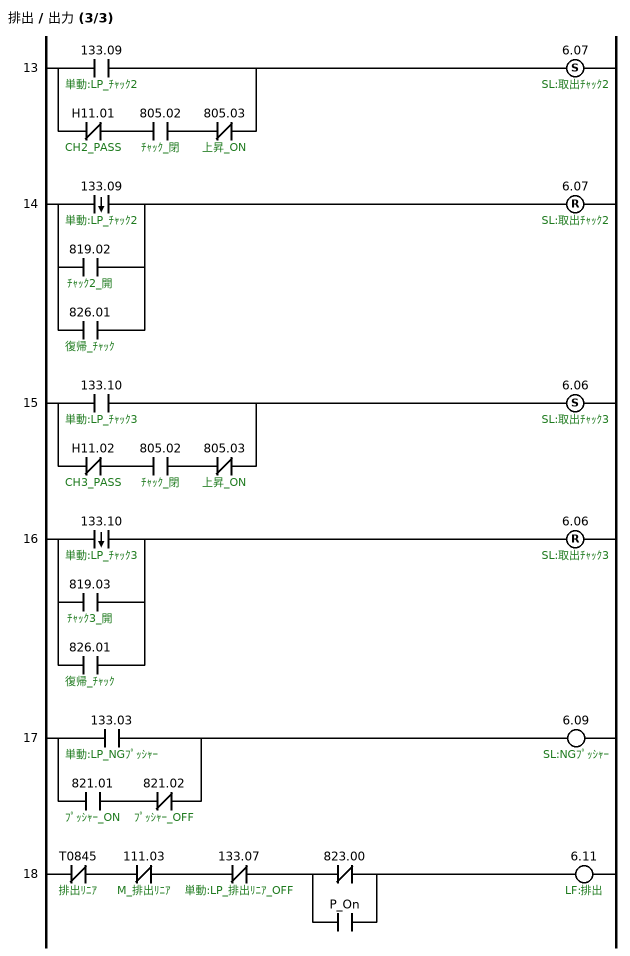
; [picture p192: 排出 / 出力, rungs 13-18]
; rung 13
LD 133.09  ; 単動:LP_ﾁｬｯｸ2
LDNOT H11.01  ; CH2_PASS
AND 805.02  ; ﾁｬｯｸ_閉
ANDNOT 805.03  ; 上昇_ON
ORLD
SET 6.07  ; SL:取出ﾁｬｯｸ2
; rung 14
%LD 133.09  ; 単動:LP_ﾁｬｯｸ2
OR 819.02  ; ﾁｬｯｸ2_開
OR 826.01  ; 復帰_ﾁｬｯｸ
RSET 6.07  ; SL:取出ﾁｬｯｸ2
; rung 15
LD 133.10  ; 単動:LP_ﾁｬｯｸ3
LDNOT H11.02  ; CH3_PASS
AND 805.02  ; ﾁｬｯｸ_閉
ANDNOT 805.03  ; 上昇_ON
ORLD
SET 6.06  ; SL:取出ﾁｬｯｸ3
; rung 16
%LD 133.10  ; 単動:LP_ﾁｬｯｸ3
OR 819.03  ; ﾁｬｯｸ3_開
OR 826.01  ; 復帰_ﾁｬｯｸ
RSET 6.06  ; SL:取出ﾁｬｯｸ3
; rung 17
LD 133.03  ; 単動:LP_NGﾌﾟｯｼｬｰ
LD 821.01  ; ﾌﾟｯｼｬｰ_ON
ANDNOT 821.02  ; ﾌﾟｯｼｬｰ_OFF
ORLD
OUT 6.09  ; SL:NGﾌﾟｯｼｬｰ
; rung 18
LDNOT T0845  ; 排出ﾘﾆｱ
ANDNOT 111.03  ; M_排出ﾘﾆｱ
ANDNOT 133.07  ; 単動:LP_排出ﾘﾆｱ_OFF
LDNOT 823.00
OR P_On
ANDLD
OUT 6.11  ; LF:排出

### Section ｴﾗｰ

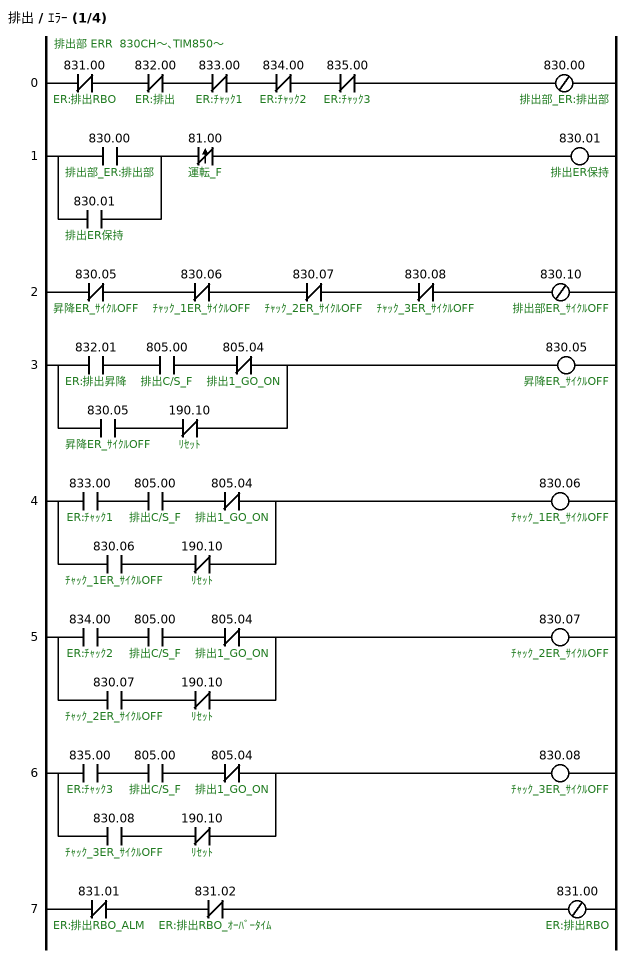
; rung 0: 排出部 ERR  830CH～､TIM850～
LDNOT 831.00  ; ER:排出RBO
ANDNOT 832.00  ; ER:排出
ANDNOT 833.00  ; ER:ﾁｬｯｸ1
ANDNOT 834.00  ; ER:ﾁｬｯｸ2
ANDNOT 835.00  ; ER:ﾁｬｯｸ3
OUTNOT 830.00  ; 排出部_ER:排出部
; rung 1
LD 830.00  ; 排出部_ER:排出部
OR 830.01  ; 排出ER保持
@ANDNOT 81.00  ; 運転_F
OUT 830.01  ; 排出ER保持
; rung 2
LDNOT 830.05  ; 昇降ER_ｻｲｸﾙOFF
ANDNOT 830.06  ; ﾁｬｯｸ_1ER_ｻｲｸﾙOFF
ANDNOT 830.07  ; ﾁｬｯｸ_2ER_ｻｲｸﾙOFF
ANDNOT 830.08  ; ﾁｬｯｸ_3ER_ｻｲｸﾙOFF
OUTNOT 830.10  ; 排出部ER_ｻｲｸﾙOFF
; rung 3
LD 832.01  ; ER:排出昇降
AND 805.00  ; 排出C/S_F
ANDNOT 805.04  ; 排出1_GO_ON
LD 830.05  ; 昇降ER_ｻｲｸﾙOFF
ANDNOT 190.10  ; ﾘｾｯﾄ
ORLD
OUT 830.05  ; 昇降ER_ｻｲｸﾙOFF
; rung 4
LD 833.00  ; ER:ﾁｬｯｸ1
AND 805.00  ; 排出C/S_F
ANDNOT 805.04  ; 排出1_GO_ON
LD 830.06  ; ﾁｬｯｸ_1ER_ｻｲｸﾙOFF
ANDNOT 190.10  ; ﾘｾｯﾄ
ORLD
OUT 830.06  ; ﾁｬｯｸ_1ER_ｻｲｸﾙOFF
; rung 5
LD 834.00  ; ER:ﾁｬｯｸ2
AND 805.00  ; 排出C/S_F
ANDNOT 805.04  ; 排出1_GO_ON
LD 830.07  ; ﾁｬｯｸ_2ER_ｻｲｸﾙOFF
ANDNOT 190.10  ; ﾘｾｯﾄ
ORLD
OUT 830.07  ; ﾁｬｯｸ_2ER_ｻｲｸﾙOFF
; rung 6
LD 835.00  ; ER:ﾁｬｯｸ3
AND 805.00  ; 排出C/S_F
ANDNOT 805.04  ; 排出1_GO_ON
LD 830.08  ; ﾁｬｯｸ_3ER_ｻｲｸﾙOFF
ANDNOT 190.10  ; ﾘｾｯﾄ
ORLD
OUT 830.08  ; ﾁｬｯｸ_3ER_ｻｲｸﾙOFF
; rung 7
LDNOT 831.01  ; ER:排出RBO_ALM
ANDNOT 831.02  ; ER:排出RBO_ｵｰﾊﾞｰﾀｲﾑ
OUTNOT 831.00  ; ER:排出RBO

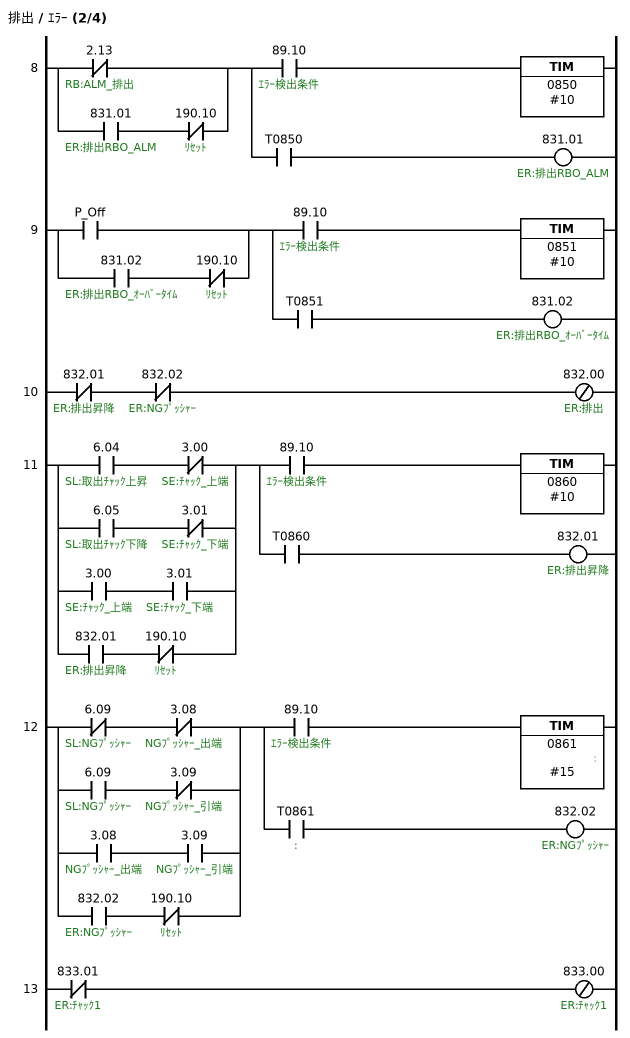
; rung 8
LDNOT 2.13  ; RB:ALM_排出
LD 831.01  ; ER:排出RBO_ALM
ANDNOT 190.10  ; ﾘｾｯﾄ
ORLD
OUT TR0
AND 89.10  ; ｴﾗｰ検出条件
TIM 0850 #10
LD TR0
AND T0850
OUT 831.01  ; ER:排出RBO_ALM
; rung 9
LD P_Off
LD 831.02  ; ER:排出RBO_ｵｰﾊﾞｰﾀｲﾑ
ANDNOT 190.10  ; ﾘｾｯﾄ
ORLD
OUT TR0
AND 89.10  ; ｴﾗｰ検出条件
TIM 0851 #10
LD TR0
AND T0851
OUT 831.02  ; ER:排出RBO_ｵｰﾊﾞｰﾀｲﾑ
; rung 10
LDNOT 832.01  ; ER:排出昇降
ANDNOT 832.02  ; ER:NGﾌﾟｯｼｬｰ
OUTNOT 832.00  ; ER:排出
; rung 11
LD 6.04  ; SL:取出ﾁｬｯｸ上昇
ANDNOT 3.00  ; SE:ﾁｬｯｸ_上端
LD 6.05  ; SL:取出ﾁｬｯｸ下降
ANDNOT 3.01  ; SE:ﾁｬｯｸ_下端
ORLD
LD 3.00  ; SE:ﾁｬｯｸ_上端
AND 3.01  ; SE:ﾁｬｯｸ_下端
ORLD
LD 832.01  ; ER:排出昇降
ANDNOT 190.10  ; ﾘｾｯﾄ
ORLD
OUT TR0
AND 89.10  ; ｴﾗｰ検出条件
TIM 0860 #10
LD TR0
AND T0860
OUT 832.01  ; ER:排出昇降
; rung 12
LDNOT 6.09  ; SL:NGﾌﾟｯｼｬｰ
ANDNOT 3.08  ; NGﾌﾟｯｼｬｰ_出端
LD 6.09  ; SL:NGﾌﾟｯｼｬｰ
ANDNOT 3.09  ; NGﾌﾟｯｼｬｰ_引端
ORLD
LD 3.08  ; NGﾌﾟｯｼｬｰ_出端
AND 3.09  ; NGﾌﾟｯｼｬｰ_引端
ORLD
LD 832.02  ; ER:NGﾌﾟｯｼｬｰ
ANDNOT 190.10  ; ﾘｾｯﾄ
ORLD
OUT TR0
AND 89.10  ; ｴﾗｰ検出条件
TIM 0861 #15  ; :
LD TR0
AND T0861  ; :
OUT 832.02  ; ER:NGﾌﾟｯｼｬｰ
; rung 13
LDNOT 833.01  ; ER:ﾁｬｯｸ1
OUTNOT 833.00  ; ER:ﾁｬｯｸ1

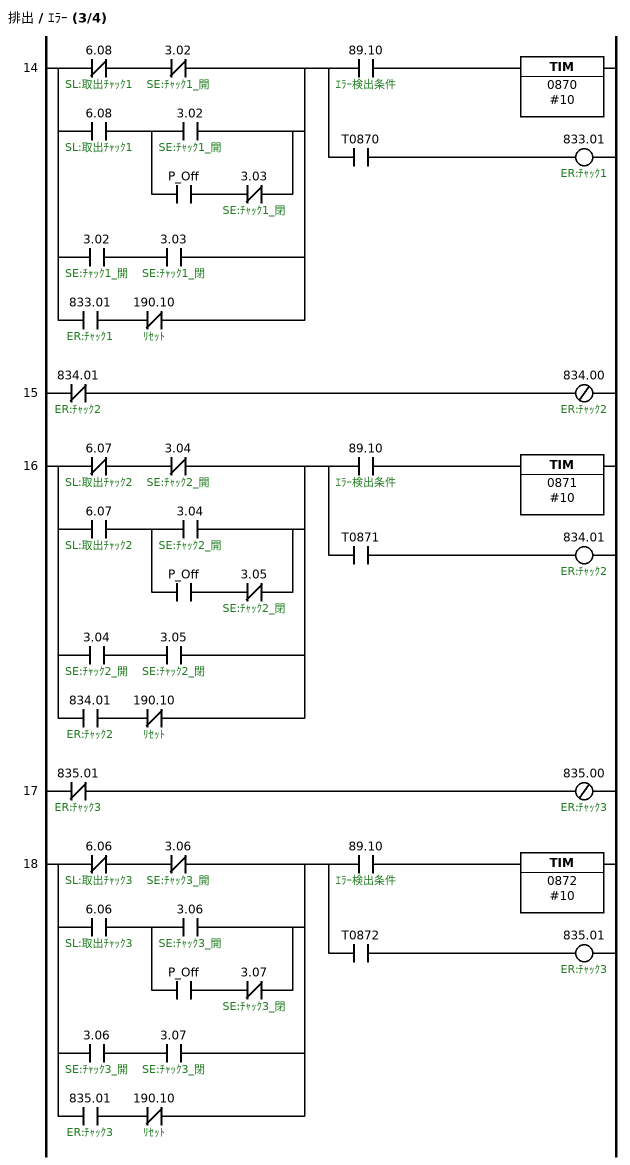
; rung 14
LDNOT 6.08  ; SL:取出ﾁｬｯｸ1
ANDNOT 3.02  ; SE:ﾁｬｯｸ1_開
LD 6.08  ; SL:取出ﾁｬｯｸ1
LD 3.02  ; SE:ﾁｬｯｸ1_開
LD P_Off
ANDNOT 3.03  ; SE:ﾁｬｯｸ1_閉
ORLD
ANDLD
ORLD
LD 3.02  ; SE:ﾁｬｯｸ1_開
AND 3.03  ; SE:ﾁｬｯｸ1_閉
ORLD
LD 833.01  ; ER:ﾁｬｯｸ1
ANDNOT 190.10  ; ﾘｾｯﾄ
ORLD
OUT TR0
AND 89.10  ; ｴﾗｰ検出条件
TIM 0870 #10
LD TR0
AND T0870
OUT 833.01  ; ER:ﾁｬｯｸ1
; rung 15
LDNOT 834.01  ; ER:ﾁｬｯｸ2
OUTNOT 834.00  ; ER:ﾁｬｯｸ2
; rung 16
LDNOT 6.07  ; SL:取出ﾁｬｯｸ2
ANDNOT 3.04  ; SE:ﾁｬｯｸ2_開
LD 6.07  ; SL:取出ﾁｬｯｸ2
LD 3.04  ; SE:ﾁｬｯｸ2_開
LD P_Off
ANDNOT 3.05  ; SE:ﾁｬｯｸ2_閉
ORLD
ANDLD
ORLD
LD 3.04  ; SE:ﾁｬｯｸ2_開
AND 3.05  ; SE:ﾁｬｯｸ2_閉
ORLD
LD 834.01  ; ER:ﾁｬｯｸ2
ANDNOT 190.10  ; ﾘｾｯﾄ
ORLD
OUT TR0
AND 89.10  ; ｴﾗｰ検出条件
TIM 0871 #10
LD TR0
AND T0871
OUT 834.01  ; ER:ﾁｬｯｸ2
; rung 17
LDNOT 835.01  ; ER:ﾁｬｯｸ3
OUTNOT 835.00  ; ER:ﾁｬｯｸ3
; rung 18
LDNOT 6.06  ; SL:取出ﾁｬｯｸ3
ANDNOT 3.06  ; SE:ﾁｬｯｸ3_開
LD 6.06  ; SL:取出ﾁｬｯｸ3
LD 3.06  ; SE:ﾁｬｯｸ3_開
LD P_Off
ANDNOT 3.07  ; SE:ﾁｬｯｸ3_閉
ORLD
ANDLD
ORLD
LD 3.06  ; SE:ﾁｬｯｸ3_開
AND 3.07  ; SE:ﾁｬｯｸ3_閉
ORLD
LD 835.01  ; ER:ﾁｬｯｸ3
ANDNOT 190.10  ; ﾘｾｯﾄ
ORLD
OUT TR0
AND 89.10  ; ｴﾗｰ検出条件
TIM 0872 #10
LD TR0
AND T0872
OUT 835.01  ; ER:ﾁｬｯｸ3

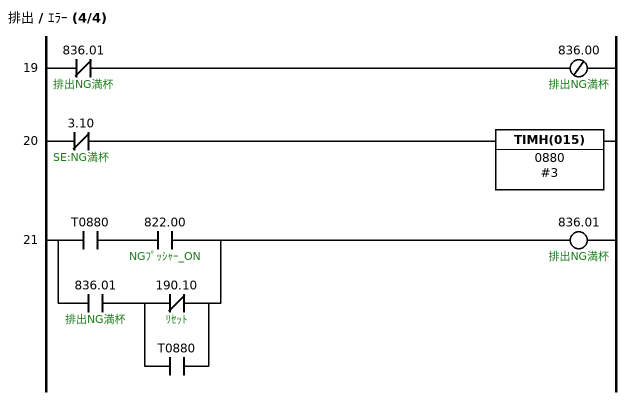
; rung 19
LDNOT 836.01  ; 排出NG満杯
OUTNOT 836.00  ; 排出NG満杯
; rung 20
LDNOT 3.10  ; SE:NG満杯
TIMH(015) 0880 #3
; rung 21
LD T0880
AND 822.00  ; NGﾌﾟｯｼｬｰ_ON
LD 836.01  ; 排出NG満杯
LDNOT 190.10  ; ﾘｾｯﾄ
OR T0880
ANDLD
ORLD
OUT 836.01  ; 排出NG満杯

### Section END
; rung 0
END(001)

## Program ﾃﾞｰﾀ収集 (cyclic task 8)

### Section 通信ST

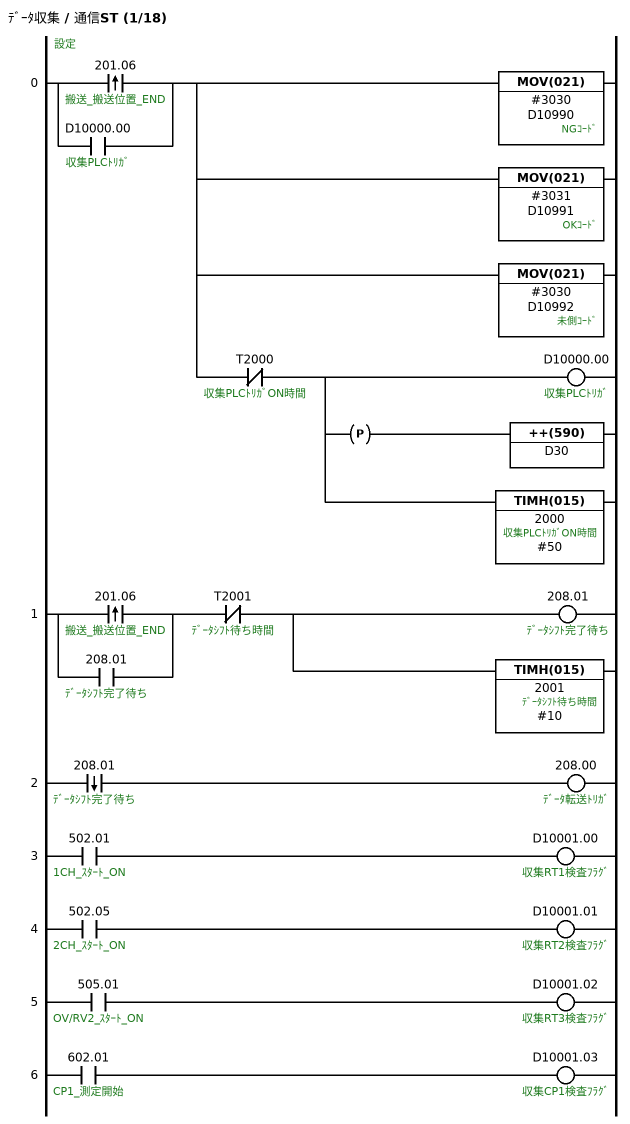
; rung 0: 設定
@LD 201.06  ; 搬送_搬送位置_END
OR D10000.00  ; 収集PLCﾄﾘｶﾞ
MOV(021) #3030 D10990  ; NGｺｰﾄﾞ
MOV(021) #3031 D10991  ; OKｺｰﾄﾞ
MOV(021) #3030 D10992  ; 未側ｺｰﾄﾞ
ANDNOT T2000  ; 収集PLCﾄﾘｶﾞON時間
OUT TR0
OUT D10000.00  ; 収集PLCﾄﾘｶﾞ
UP(521)
++(590) D30
LD TR0
TIMH(015) 2000 #50  ; 収集PLCﾄﾘｶﾞON時間
; rung 1
@LD 201.06  ; 搬送_搬送位置_END
OR 208.01  ; ﾃﾞｰﾀｼﾌﾄ完了待ち
ANDNOT T2001  ; ﾃﾞｰﾀｼﾌﾄ待ち時間
OUT 208.01  ; ﾃﾞｰﾀｼﾌﾄ完了待ち
TIMH(015) 2001 #10  ; ﾃﾞｰﾀｼﾌﾄ待ち時間
; rung 2
%LD 208.01  ; ﾃﾞｰﾀｼﾌﾄ完了待ち
OUT 208.00  ; ﾃﾞｰﾀ転送ﾄﾘｶﾞ
; rung 3
LD 502.01  ; 1CH_ｽﾀｰﾄ_ON
OUT D10001.00  ; 収集RT1検査ﾌﾗｸﾞ
; rung 4
LD 502.05  ; 2CH_ｽﾀｰﾄ_ON
OUT D10001.01  ; 収集RT2検査ﾌﾗｸﾞ
; rung 5
LD 505.01  ; OV/RV2_ｽﾀｰﾄ_ON
OUT D10001.02  ; 収集RT3検査ﾌﾗｸﾞ
; rung 6
LD 602.01  ; CP1_測定開始
OUT D10001.03  ; 収集CP1検査ﾌﾗｸﾞ

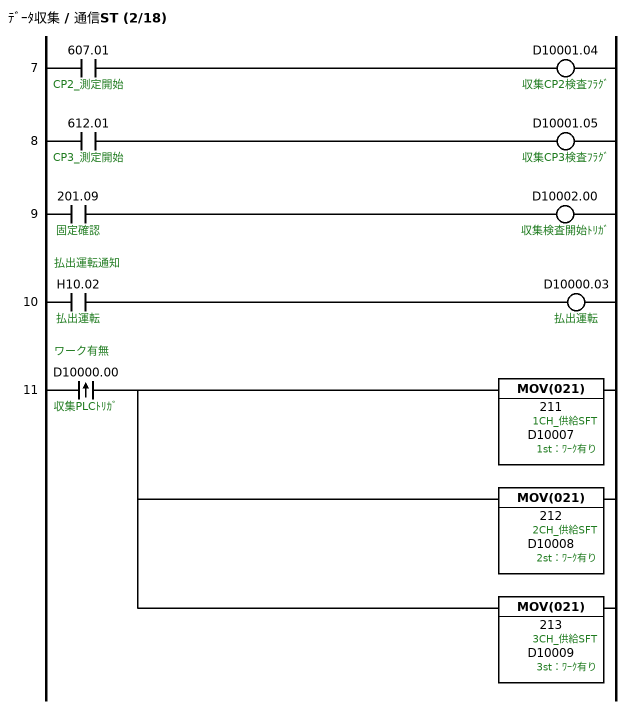
; rung 7
LD 607.01  ; CP2_測定開始
OUT D10001.04  ; 収集CP2検査ﾌﾗｸﾞ
; rung 8
LD 612.01  ; CP3_測定開始
OUT D10001.05  ; 収集CP3検査ﾌﾗｸﾞ
; rung 9
LD 201.09  ; 固定確認
OUT D10002.00  ; 収集検査開始ﾄﾘｶﾞ
; rung 10: 払出運転通知
LD H10.02  ; 払出運転
OUT D10000.03  ; 払出運転
; rung 11: ワーク有無
@LD D10000.00  ; 収集PLCﾄﾘｶﾞ
MOV(021) 211 D10007  ; 1CH_供給SFT, 1st：ﾜｰｸ有り
MOV(021) 212 D10008  ; 2CH_供給SFT, 2st：ﾜｰｸ有り
MOV(021) 213 D10009  ; 3CH_供給SFT, 3st：ﾜｰｸ有り

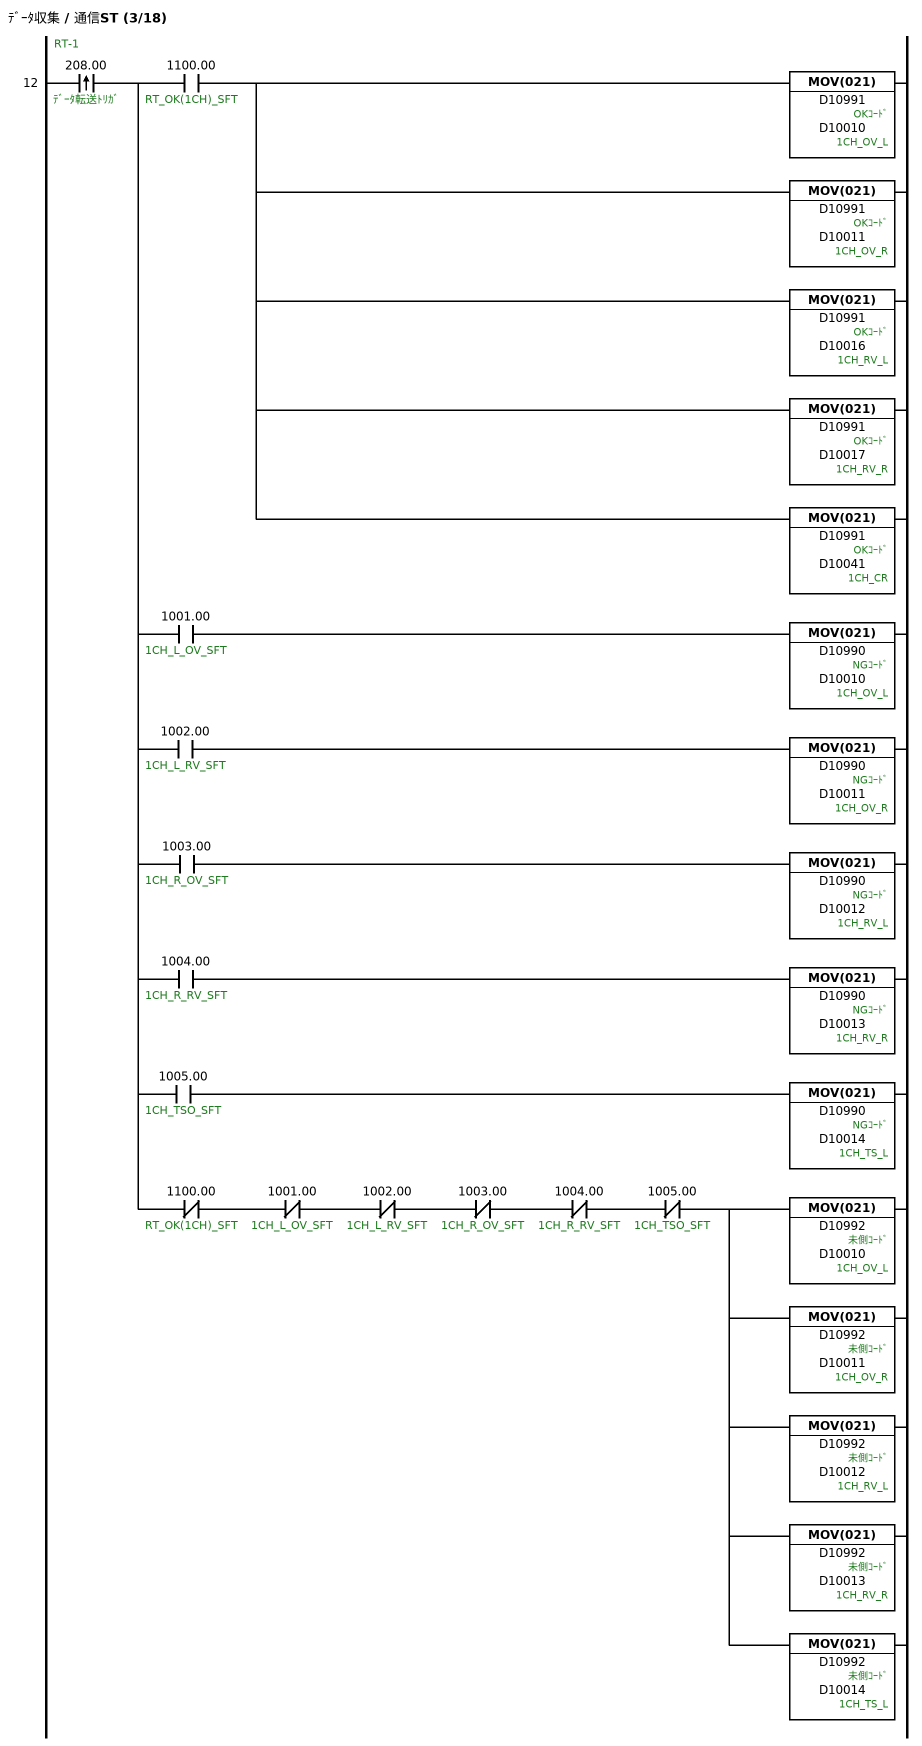
; rung 12: RT-1
@LD 208.00  ; ﾃﾞｰﾀ転送ﾄﾘｶﾞ
OUT TR0
AND 1100.00  ; RT_OK(1CH)_SFT
MOV(021) D10991 D10010  ; OKｺｰﾄﾞ, 1CH_OV_L
MOV(021) D10991 D10011  ; OKｺｰﾄﾞ, 1CH_OV_R
MOV(021) D10991 D10016  ; OKｺｰﾄﾞ, 1CH_RV_L
MOV(021) D10991 D10017  ; OKｺｰﾄﾞ, 1CH_RV_R
MOV(021) D10991 D10041  ; OKｺｰﾄﾞ, 1CH_CR
LD TR0
AND 1001.00  ; 1CH_L_OV_SFT
MOV(021) D10990 D10010  ; NGｺｰﾄﾞ, 1CH_OV_L
LD TR0
AND 1002.00  ; 1CH_L_RV_SFT
MOV(021) D10990 D10011  ; NGｺｰﾄﾞ, 1CH_OV_R
LD TR0
AND 1003.00  ; 1CH_R_OV_SFT
MOV(021) D10990 D10012  ; NGｺｰﾄﾞ, 1CH_RV_L
LD TR0
AND 1004.00  ; 1CH_R_RV_SFT
MOV(021) D10990 D10013  ; NGｺｰﾄﾞ, 1CH_RV_R
LD TR0
AND 1005.00  ; 1CH_TSO_SFT
MOV(021) D10990 D10014  ; NGｺｰﾄﾞ, 1CH_TS_L
LD TR0
ANDNOT 1100.00  ; RT_OK(1CH)_SFT
ANDNOT 1001.00  ; 1CH_L_OV_SFT
ANDNOT 1002.00  ; 1CH_L_RV_SFT
ANDNOT 1003.00  ; 1CH_R_OV_SFT
ANDNOT 1004.00  ; 1CH_R_RV_SFT
ANDNOT 1005.00  ; 1CH_TSO_SFT
MOV(021) D10992 D10010  ; 未側ｺｰﾄﾞ, 1CH_OV_L
MOV(021) D10992 D10011  ; 未側ｺｰﾄﾞ, 1CH_OV_R
MOV(021) D10992 D10012  ; 未側ｺｰﾄﾞ, 1CH_RV_L
MOV(021) D10992 D10013  ; 未側ｺｰﾄﾞ, 1CH_RV_R
MOV(021) D10992 D10014  ; 未側ｺｰﾄﾞ, 1CH_TS_L

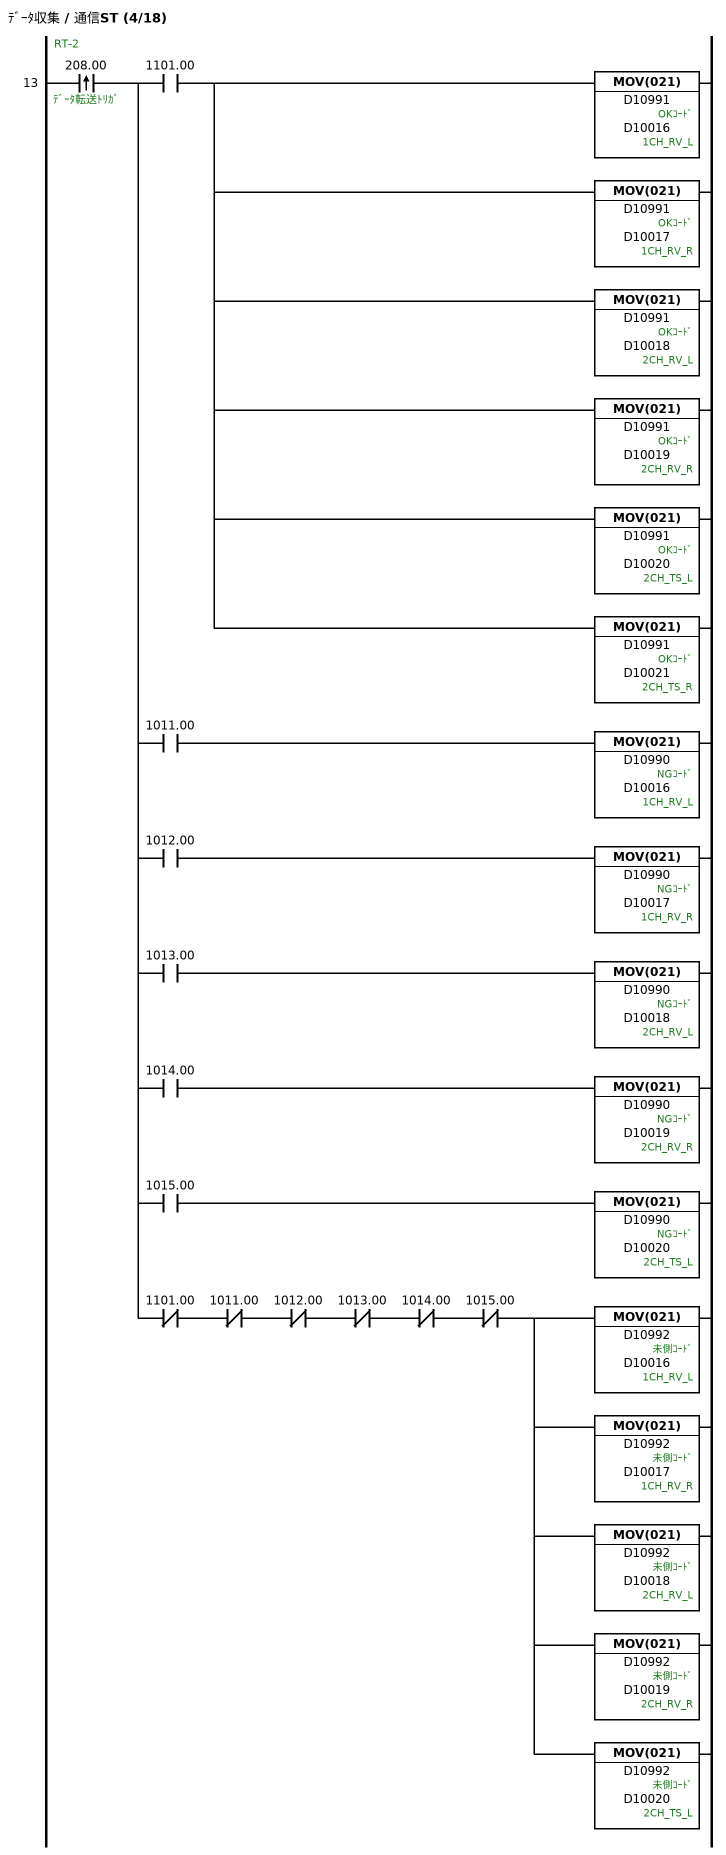
; rung 13: RT-2
@LD 208.00  ; ﾃﾞｰﾀ転送ﾄﾘｶﾞ
OUT TR0
AND 1101.00
MOV(021) D10991 D10016  ; OKｺｰﾄﾞ, 1CH_RV_L
MOV(021) D10991 D10017  ; OKｺｰﾄﾞ, 1CH_RV_R
MOV(021) D10991 D10018  ; OKｺｰﾄﾞ, 2CH_RV_L
MOV(021) D10991 D10019  ; OKｺｰﾄﾞ, 2CH_RV_R
MOV(021) D10991 D10020  ; OKｺｰﾄﾞ, 2CH_TS_L
MOV(021) D10991 D10021  ; OKｺｰﾄﾞ, 2CH_TS_R
LD TR0
AND 1011.00
MOV(021) D10990 D10016  ; NGｺｰﾄﾞ, 1CH_RV_L
LD TR0
AND 1012.00
MOV(021) D10990 D10017  ; NGｺｰﾄﾞ, 1CH_RV_R
LD TR0
AND 1013.00
MOV(021) D10990 D10018  ; NGｺｰﾄﾞ, 2CH_RV_L
LD TR0
AND 1014.00
MOV(021) D10990 D10019  ; NGｺｰﾄﾞ, 2CH_RV_R
LD TR0
AND 1015.00
MOV(021) D10990 D10020  ; NGｺｰﾄﾞ, 2CH_TS_L
LD TR0
ANDNOT 1101.00
ANDNOT 1011.00
ANDNOT 1012.00
ANDNOT 1013.00
ANDNOT 1014.00
ANDNOT 1015.00
MOV(021) D10992 D10016  ; 未側ｺｰﾄﾞ, 1CH_RV_L
MOV(021) D10992 D10017  ; 未側ｺｰﾄﾞ, 1CH_RV_R
MOV(021) D10992 D10018  ; 未側ｺｰﾄﾞ, 2CH_RV_L
MOV(021) D10992 D10019  ; 未側ｺｰﾄﾞ, 2CH_RV_R
MOV(021) D10992 D10020  ; 未側ｺｰﾄﾞ, 2CH_TS_L

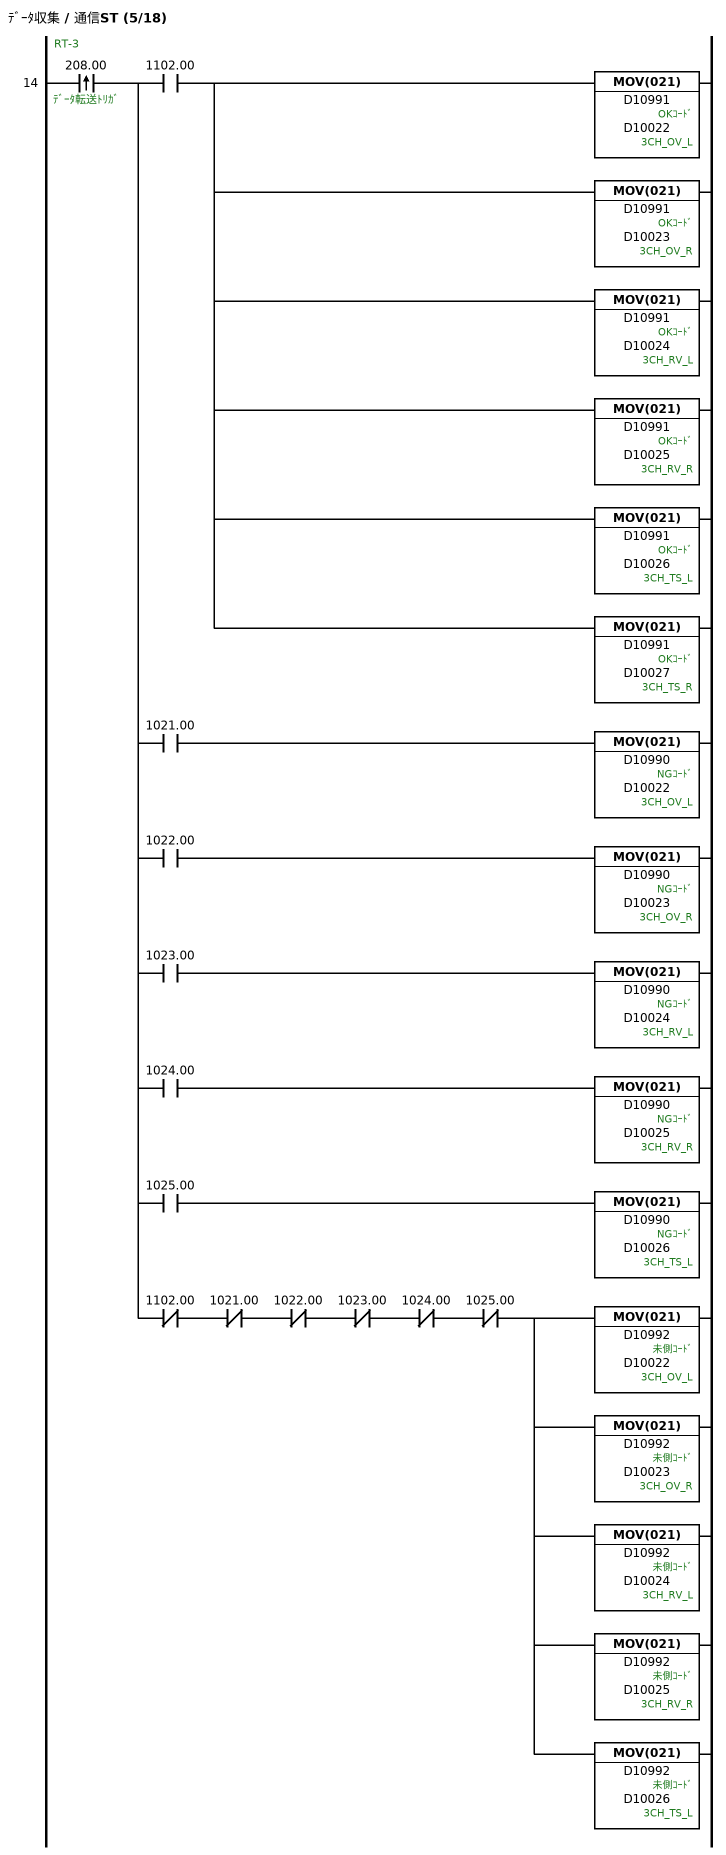
; rung 14: RT-3
@LD 208.00  ; ﾃﾞｰﾀ転送ﾄﾘｶﾞ
OUT TR0
AND 1102.00
MOV(021) D10991 D10022  ; OKｺｰﾄﾞ, 3CH_OV_L
MOV(021) D10991 D10023  ; OKｺｰﾄﾞ, 3CH_OV_R
MOV(021) D10991 D10024  ; OKｺｰﾄﾞ, 3CH_RV_L
MOV(021) D10991 D10025  ; OKｺｰﾄﾞ, 3CH_RV_R
MOV(021) D10991 D10026  ; OKｺｰﾄﾞ, 3CH_TS_L
MOV(021) D10991 D10027  ; OKｺｰﾄﾞ, 3CH_TS_R
LD TR0
AND 1021.00
MOV(021) D10990 D10022  ; NGｺｰﾄﾞ, 3CH_OV_L
LD TR0
AND 1022.00
MOV(021) D10990 D10023  ; NGｺｰﾄﾞ, 3CH_OV_R
LD TR0
AND 1023.00
MOV(021) D10990 D10024  ; NGｺｰﾄﾞ, 3CH_RV_L
LD TR0
AND 1024.00
MOV(021) D10990 D10025  ; NGｺｰﾄﾞ, 3CH_RV_R
LD TR0
AND 1025.00
MOV(021) D10990 D10026  ; NGｺｰﾄﾞ, 3CH_TS_L
LD TR0
ANDNOT 1102.00
ANDNOT 1021.00
ANDNOT 1022.00
ANDNOT 1023.00
ANDNOT 1024.00
ANDNOT 1025.00
MOV(021) D10992 D10022  ; 未側ｺｰﾄﾞ, 3CH_OV_L
MOV(021) D10992 D10023  ; 未側ｺｰﾄﾞ, 3CH_OV_R
MOV(021) D10992 D10024  ; 未側ｺｰﾄﾞ, 3CH_RV_L
MOV(021) D10992 D10025  ; 未側ｺｰﾄﾞ, 3CH_RV_R
MOV(021) D10992 D10026  ; 未側ｺｰﾄﾞ, 3CH_TS_L

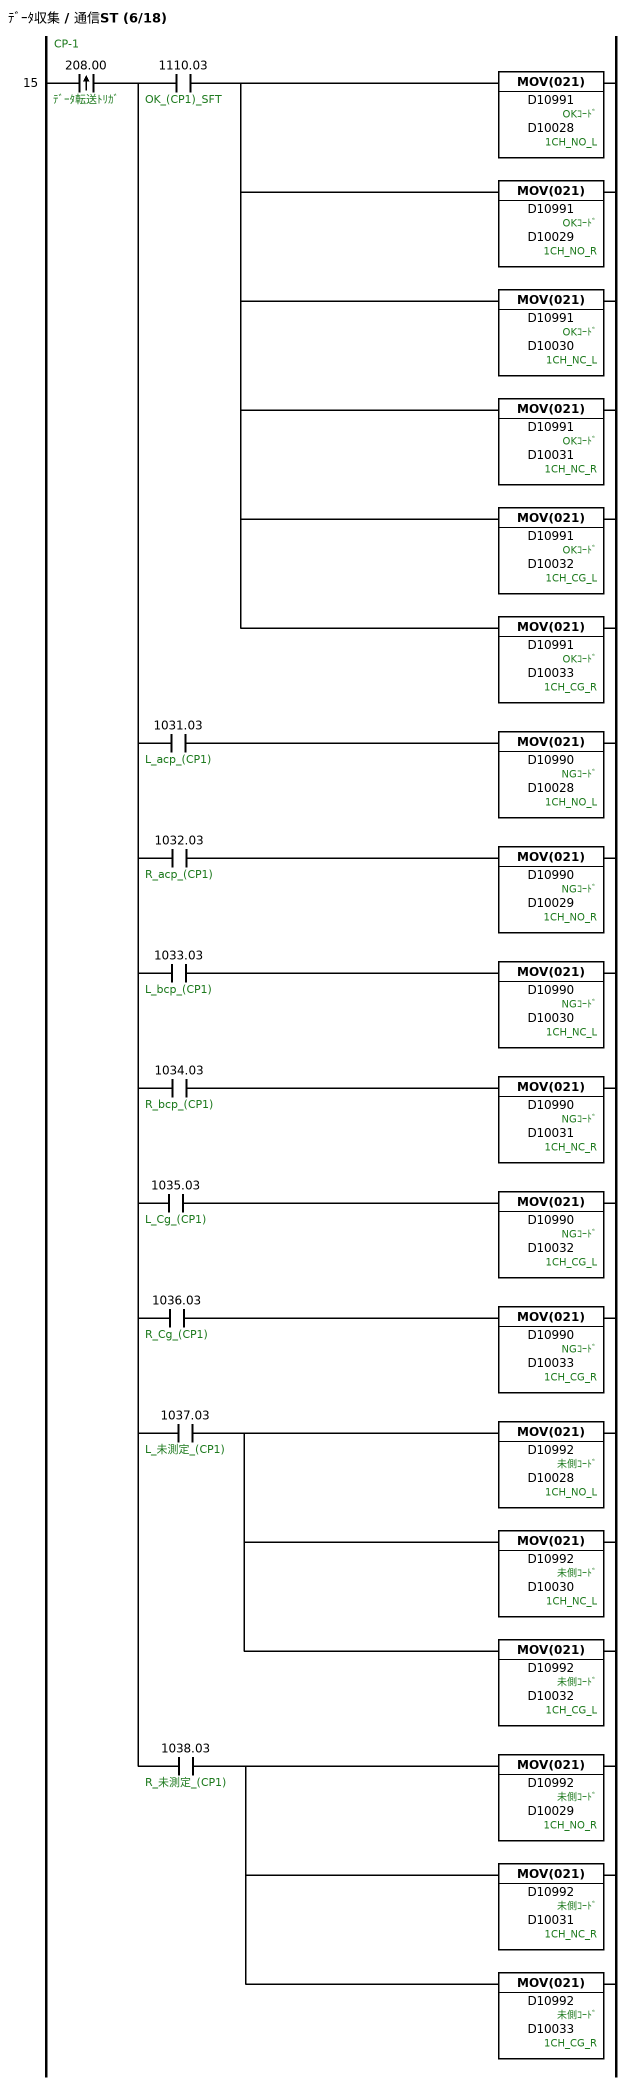
; rung 15: CP-1
@LD 208.00  ; ﾃﾞｰﾀ転送ﾄﾘｶﾞ
OUT TR0
AND 1110.03  ; OK_(CP1)_SFT
MOV(021) D10991 D10028  ; OKｺｰﾄﾞ, 1CH_NO_L
MOV(021) D10991 D10029  ; OKｺｰﾄﾞ, 1CH_NO_R
MOV(021) D10991 D10030  ; OKｺｰﾄﾞ, 1CH_NC_L
MOV(021) D10991 D10031  ; OKｺｰﾄﾞ, 1CH_NC_R
MOV(021) D10991 D10032  ; OKｺｰﾄﾞ, 1CH_CG_L
MOV(021) D10991 D10033  ; OKｺｰﾄﾞ, 1CH_CG_R
LD TR0
AND 1031.03  ; L_acp_(CP1)
MOV(021) D10990 D10028  ; NGｺｰﾄﾞ, 1CH_NO_L
LD TR0
AND 1032.03  ; R_acp_(CP1)
MOV(021) D10990 D10029  ; NGｺｰﾄﾞ, 1CH_NO_R
LD TR0
AND 1033.03  ; L_bcp_(CP1)
MOV(021) D10990 D10030  ; NGｺｰﾄﾞ, 1CH_NC_L
LD TR0
AND 1034.03  ; R_bcp_(CP1)
MOV(021) D10990 D10031  ; NGｺｰﾄﾞ, 1CH_NC_R
LD TR0
AND 1035.03  ; L_Cg_(CP1)
MOV(021) D10990 D10032  ; NGｺｰﾄﾞ, 1CH_CG_L
LD TR0
AND 1036.03  ; R_Cg_(CP1)
MOV(021) D10990 D10033  ; NGｺｰﾄﾞ, 1CH_CG_R
LD TR0
AND 1037.03  ; L_未測定_(CP1)
MOV(021) D10992 D10028  ; 未側ｺｰﾄﾞ, 1CH_NO_L
MOV(021) D10992 D10030  ; 未側ｺｰﾄﾞ, 1CH_NC_L
MOV(021) D10992 D10032  ; 未側ｺｰﾄﾞ, 1CH_CG_L
LD TR0
AND 1038.03  ; R_未測定_(CP1)
MOV(021) D10992 D10029  ; 未側ｺｰﾄﾞ, 1CH_NO_R
MOV(021) D10992 D10031  ; 未側ｺｰﾄﾞ, 1CH_NC_R
MOV(021) D10992 D10033  ; 未側ｺｰﾄﾞ, 1CH_CG_R

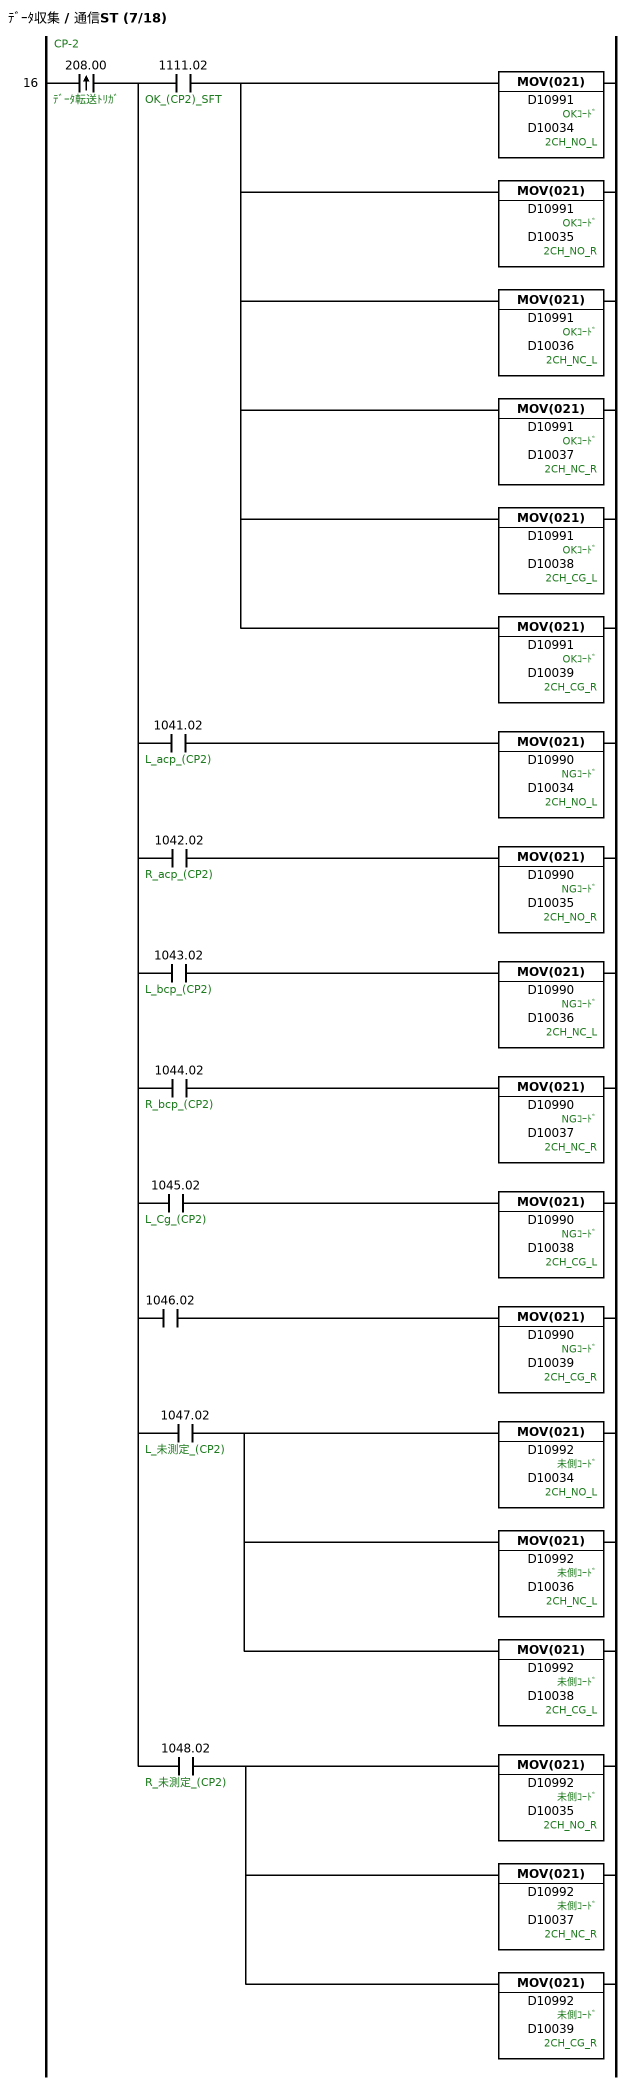
; rung 16: CP-2
@LD 208.00  ; ﾃﾞｰﾀ転送ﾄﾘｶﾞ
OUT TR0
AND 1111.02  ; OK_(CP2)_SFT
MOV(021) D10991 D10034  ; OKｺｰﾄﾞ, 2CH_NO_L
MOV(021) D10991 D10035  ; OKｺｰﾄﾞ, 2CH_NO_R
MOV(021) D10991 D10036  ; OKｺｰﾄﾞ, 2CH_NC_L
MOV(021) D10991 D10037  ; OKｺｰﾄﾞ, 2CH_NC_R
MOV(021) D10991 D10038  ; OKｺｰﾄﾞ, 2CH_CG_L
MOV(021) D10991 D10039  ; OKｺｰﾄﾞ, 2CH_CG_R
LD TR0
AND 1041.02  ; L_acp_(CP2)
MOV(021) D10990 D10034  ; NGｺｰﾄﾞ, 2CH_NO_L
LD TR0
AND 1042.02  ; R_acp_(CP2)
MOV(021) D10990 D10035  ; NGｺｰﾄﾞ, 2CH_NO_R
LD TR0
AND 1043.02  ; L_bcp_(CP2)
MOV(021) D10990 D10036  ; NGｺｰﾄﾞ, 2CH_NC_L
LD TR0
AND 1044.02  ; R_bcp_(CP2)
MOV(021) D10990 D10037  ; NGｺｰﾄﾞ, 2CH_NC_R
LD TR0
AND 1045.02  ; L_Cg_(CP2)
MOV(021) D10990 D10038  ; NGｺｰﾄﾞ, 2CH_CG_L
LD TR0
AND 1046.02
MOV(021) D10990 D10039  ; NGｺｰﾄﾞ, 2CH_CG_R
LD TR0
AND 1047.02  ; L_未測定_(CP2)
MOV(021) D10992 D10034  ; 未側ｺｰﾄﾞ, 2CH_NO_L
MOV(021) D10992 D10036  ; 未側ｺｰﾄﾞ, 2CH_NC_L
MOV(021) D10992 D10038  ; 未側ｺｰﾄﾞ, 2CH_CG_L
LD TR0
AND 1048.02  ; R_未測定_(CP2)
MOV(021) D10992 D10035  ; 未側ｺｰﾄﾞ, 2CH_NO_R
MOV(021) D10992 D10037  ; 未側ｺｰﾄﾞ, 2CH_NC_R
MOV(021) D10992 D10039  ; 未側ｺｰﾄﾞ, 2CH_CG_R

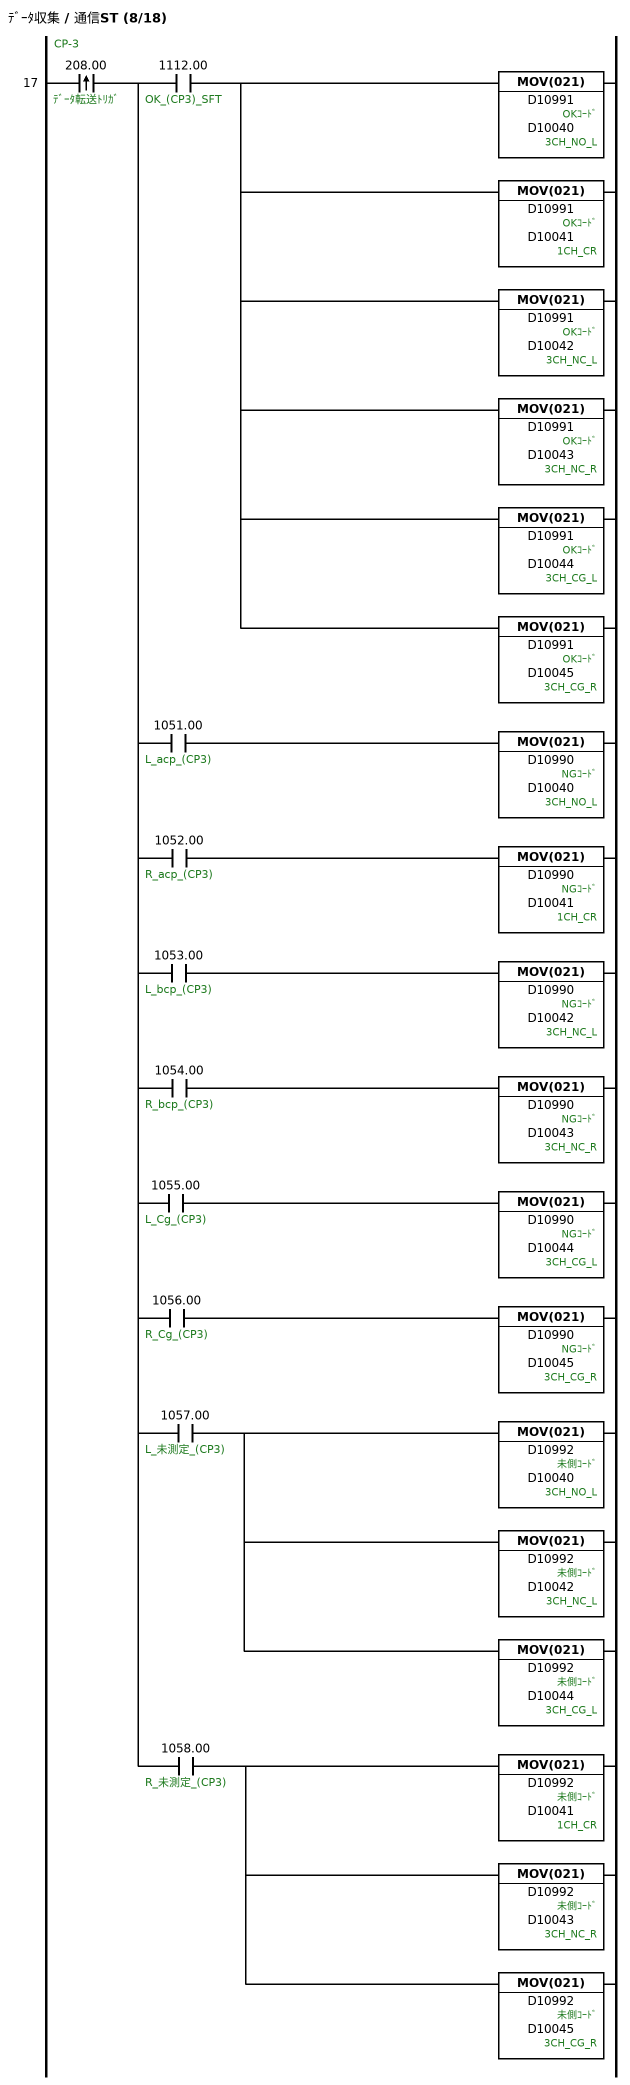
; rung 17: CP-3
@LD 208.00  ; ﾃﾞｰﾀ転送ﾄﾘｶﾞ
OUT TR0
AND 1112.00  ; OK_(CP3)_SFT
MOV(021) D10991 D10040  ; OKｺｰﾄﾞ, 3CH_NO_L
MOV(021) D10991 D10041  ; OKｺｰﾄﾞ, 1CH_CR
MOV(021) D10991 D10042  ; OKｺｰﾄﾞ, 3CH_NC_L
MOV(021) D10991 D10043  ; OKｺｰﾄﾞ, 3CH_NC_R
MOV(021) D10991 D10044  ; OKｺｰﾄﾞ, 3CH_CG_L
MOV(021) D10991 D10045  ; OKｺｰﾄﾞ, 3CH_CG_R
LD TR0
AND 1051.00  ; L_acp_(CP3)
MOV(021) D10990 D10040  ; NGｺｰﾄﾞ, 3CH_NO_L
LD TR0
AND 1052.00  ; R_acp_(CP3)
MOV(021) D10990 D10041  ; NGｺｰﾄﾞ, 1CH_CR
LD TR0
AND 1053.00  ; L_bcp_(CP3)
MOV(021) D10990 D10042  ; NGｺｰﾄﾞ, 3CH_NC_L
LD TR0
AND 1054.00  ; R_bcp_(CP3)
MOV(021) D10990 D10043  ; NGｺｰﾄﾞ, 3CH_NC_R
LD TR0
AND 1055.00  ; L_Cg_(CP3)
MOV(021) D10990 D10044  ; NGｺｰﾄﾞ, 3CH_CG_L
LD TR0
AND 1056.00  ; R_Cg_(CP3)
MOV(021) D10990 D10045  ; NGｺｰﾄﾞ, 3CH_CG_R
LD TR0
AND 1057.00  ; L_未測定_(CP3)
MOV(021) D10992 D10040  ; 未側ｺｰﾄﾞ, 3CH_NO_L
MOV(021) D10992 D10042  ; 未側ｺｰﾄﾞ, 3CH_NC_L
MOV(021) D10992 D10044  ; 未側ｺｰﾄﾞ, 3CH_CG_L
LD TR0
AND 1058.00  ; R_未測定_(CP3)
MOV(021) D10992 D10041  ; 未側ｺｰﾄﾞ, 1CH_CR
MOV(021) D10992 D10043  ; 未側ｺｰﾄﾞ, 3CH_NC_R
MOV(021) D10992 D10045  ; 未側ｺｰﾄﾞ, 3CH_CG_R

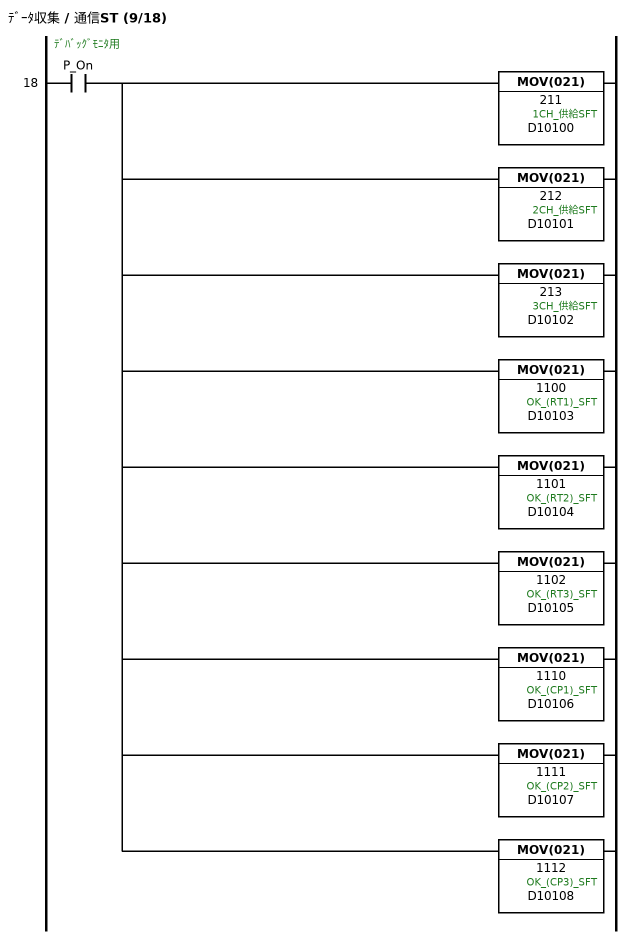
; rung 18: ﾃﾞﾊﾞｯｸﾞﾓﾆﾀ用
LD P_On
MOV(021) 211 D10100  ; 1CH_供給SFT
MOV(021) 212 D10101  ; 2CH_供給SFT
MOV(021) 213 D10102  ; 3CH_供給SFT
MOV(021) 1100 D10103  ; OK_(RT1)_SFT
MOV(021) 1101 D10104  ; OK_(RT2)_SFT
MOV(021) 1102 D10105  ; OK_(RT3)_SFT
MOV(021) 1110 D10106  ; OK_(CP1)_SFT
MOV(021) 1111 D10107  ; OK_(CP2)_SFT
MOV(021) 1112 D10108  ; OK_(CP3)_SFT

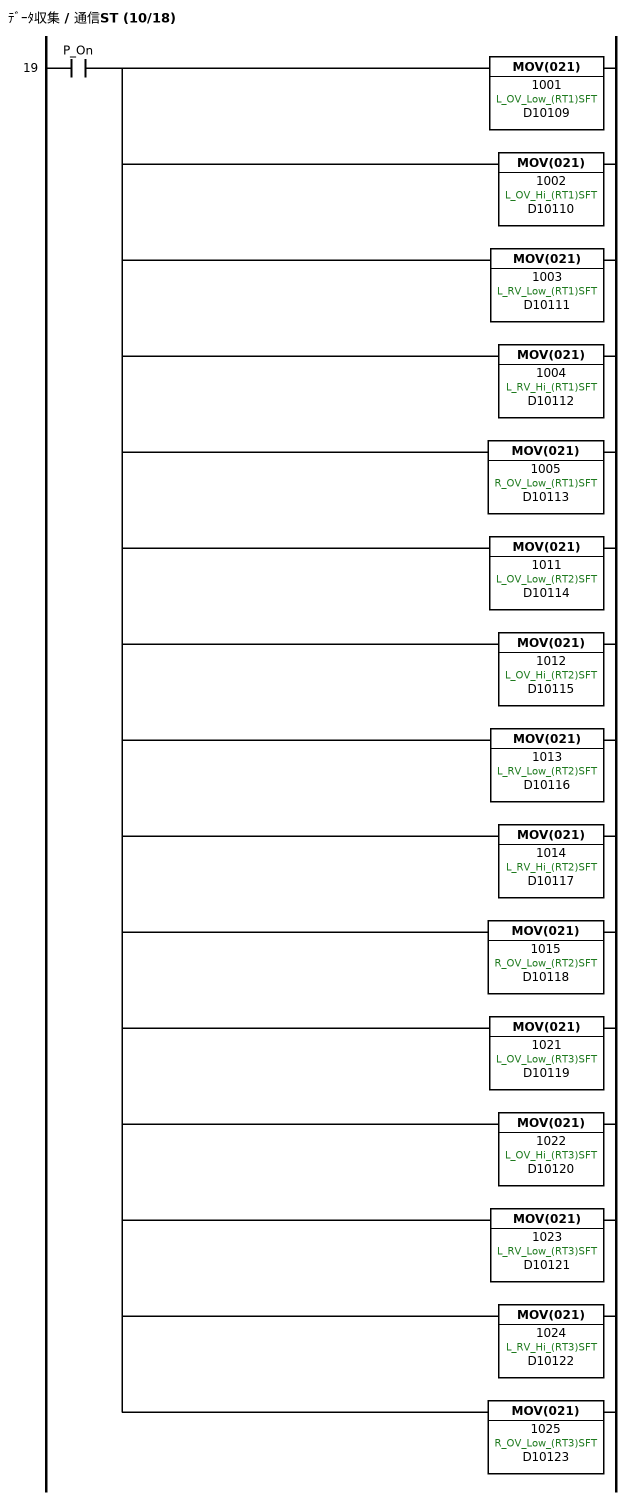
; rung 19
LD P_On
MOV(021) 1001 D10109  ; L_OV_Low_(RT1)SFT
MOV(021) 1002 D10110  ; L_OV_Hi_(RT1)SFT
MOV(021) 1003 D10111  ; L_RV_Low_(RT1)SFT
MOV(021) 1004 D10112  ; L_RV_Hi_(RT1)SFT
MOV(021) 1005 D10113  ; R_OV_Low_(RT1)SFT
MOV(021) 1011 D10114  ; L_OV_Low_(RT2)SFT
MOV(021) 1012 D10115  ; L_OV_Hi_(RT2)SFT
MOV(021) 1013 D10116  ; L_RV_Low_(RT2)SFT
MOV(021) 1014 D10117  ; L_RV_Hi_(RT2)SFT
MOV(021) 1015 D10118  ; R_OV_Low_(RT2)SFT
MOV(021) 1021 D10119  ; L_OV_Low_(RT3)SFT
MOV(021) 1022 D10120  ; L_OV_Hi_(RT3)SFT
MOV(021) 1023 D10121  ; L_RV_Low_(RT3)SFT
MOV(021) 1024 D10122  ; L_RV_Hi_(RT3)SFT
MOV(021) 1025 D10123  ; R_OV_Low_(RT3)SFT

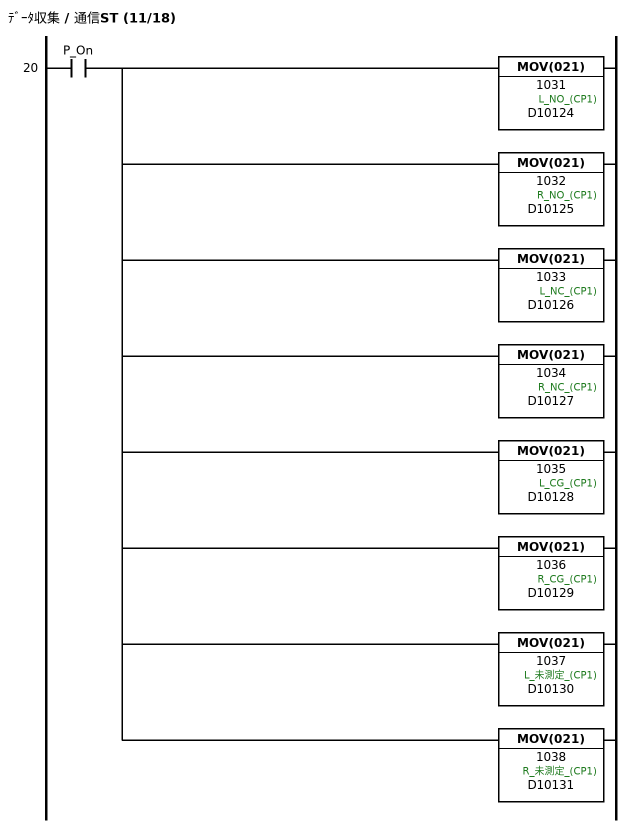
; rung 20
LD P_On
MOV(021) 1031 D10124  ; L_NO_(CP1)
MOV(021) 1032 D10125  ; R_NO_(CP1)
MOV(021) 1033 D10126  ; L_NC_(CP1)
MOV(021) 1034 D10127  ; R_NC_(CP1)
MOV(021) 1035 D10128  ; L_CG_(CP1)
MOV(021) 1036 D10129  ; R_CG_(CP1)
MOV(021) 1037 D10130  ; L_未測定_(CP1)
MOV(021) 1038 D10131  ; R_未測定_(CP1)

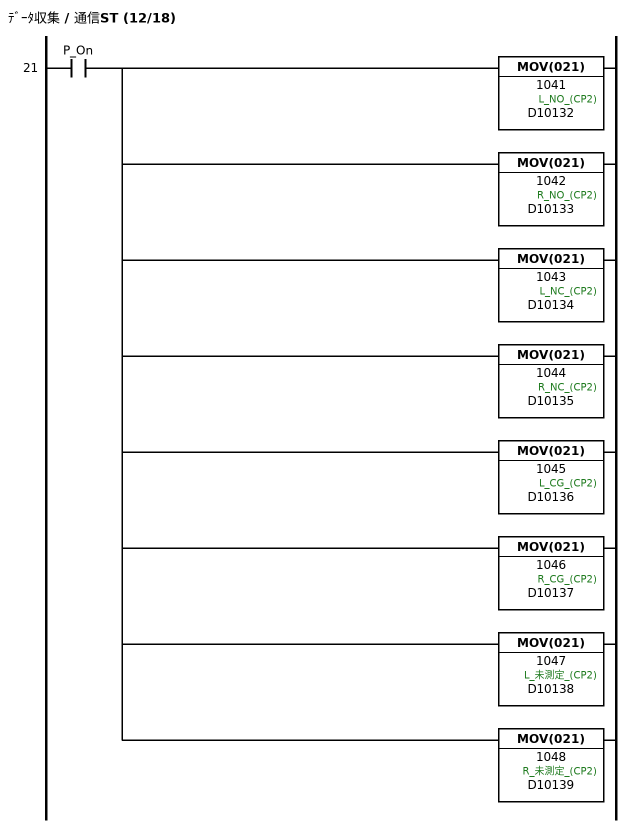
; rung 21
LD P_On
MOV(021) 1041 D10132  ; L_NO_(CP2)
MOV(021) 1042 D10133  ; R_NO_(CP2)
MOV(021) 1043 D10134  ; L_NC_(CP2)
MOV(021) 1044 D10135  ; R_NC_(CP2)
MOV(021) 1045 D10136  ; L_CG_(CP2)
MOV(021) 1046 D10137  ; R_CG_(CP2)
MOV(021) 1047 D10138  ; L_未測定_(CP2)
MOV(021) 1048 D10139  ; R_未測定_(CP2)

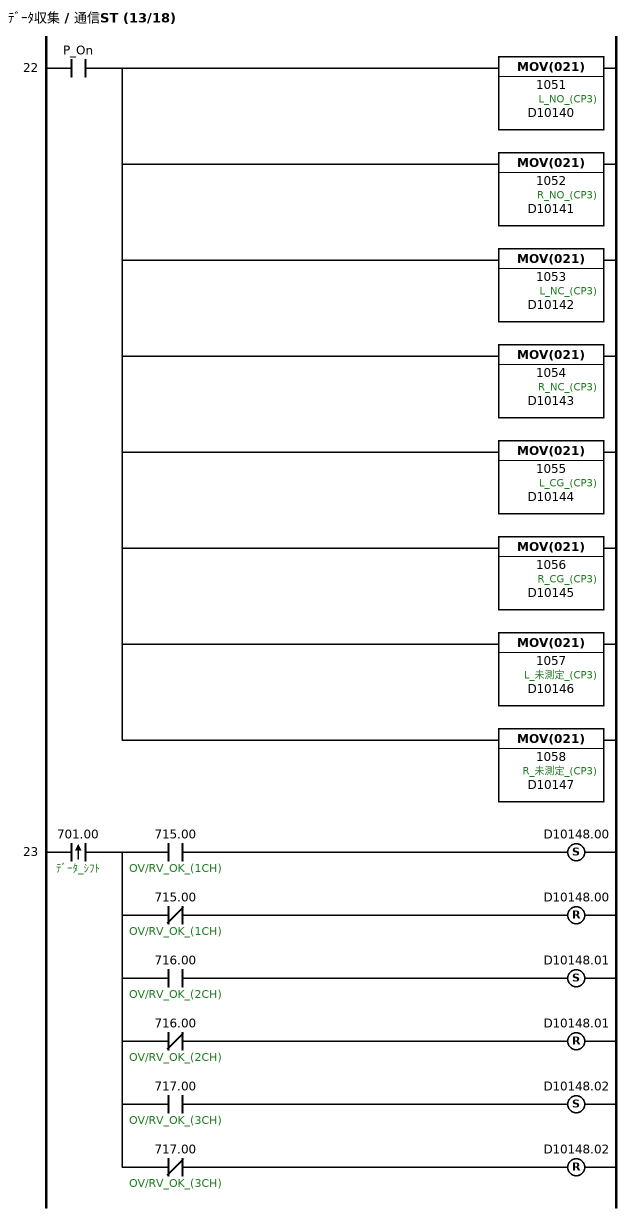
; rung 22
LD P_On
MOV(021) 1051 D10140  ; L_NO_(CP3)
MOV(021) 1052 D10141  ; R_NO_(CP3)
MOV(021) 1053 D10142  ; L_NC_(CP3)
MOV(021) 1054 D10143  ; R_NC_(CP3)
MOV(021) 1055 D10144  ; L_CG_(CP3)
MOV(021) 1056 D10145  ; R_CG_(CP3)
MOV(021) 1057 D10146  ; L_未測定_(CP3)
MOV(021) 1058 D10147  ; R_未測定_(CP3)
; rung 23
@LD 701.00  ; ﾃﾞｰﾀ_ｼﾌﾄ
OUT TR0
AND 715.00  ; OV/RV_OK_(1CH)
SET D10148.00
LD TR0
ANDNOT 715.00  ; OV/RV_OK_(1CH)
RSET D10148.00
LD TR0
AND 716.00  ; OV/RV_OK_(2CH)
SET D10148.01
LD TR0
ANDNOT 716.00  ; OV/RV_OK_(2CH)
RSET D10148.01
LD TR0
AND 717.00  ; OV/RV_OK_(3CH)
SET D10148.02
LD TR0
ANDNOT 717.00  ; OV/RV_OK_(3CH)
RSET D10148.02

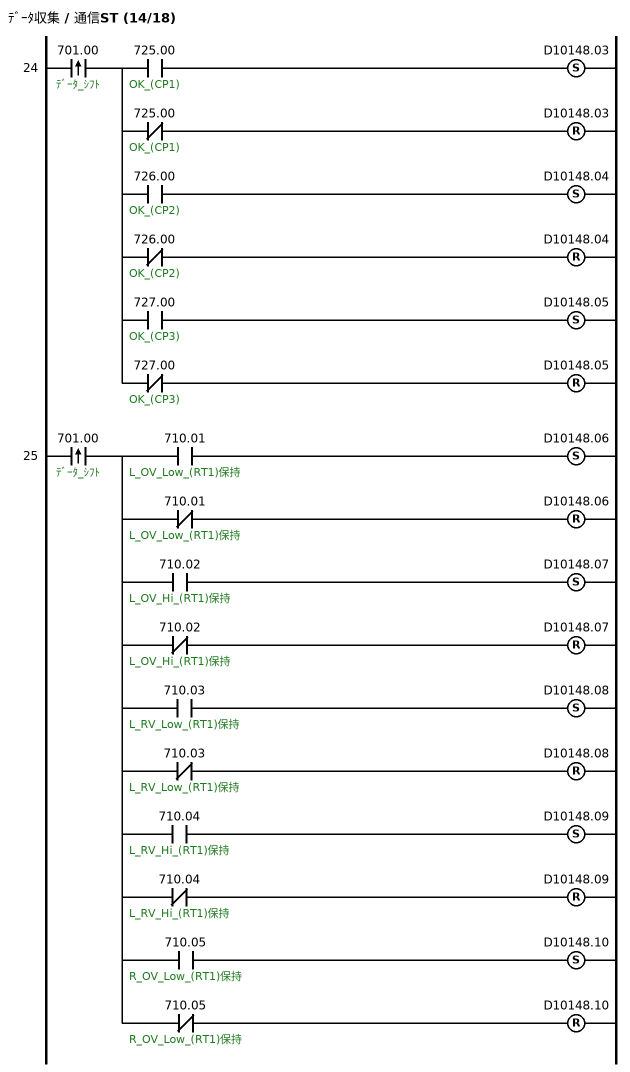
; rung 24
@LD 701.00  ; ﾃﾞｰﾀ_ｼﾌﾄ
OUT TR0
AND 725.00  ; OK_(CP1)
SET D10148.03
LD TR0
ANDNOT 725.00  ; OK_(CP1)
RSET D10148.03
LD TR0
AND 726.00  ; OK_(CP2)
SET D10148.04
LD TR0
ANDNOT 726.00  ; OK_(CP2)
RSET D10148.04
LD TR0
AND 727.00  ; OK_(CP3)
SET D10148.05
LD TR0
ANDNOT 727.00  ; OK_(CP3)
RSET D10148.05
; rung 25
@LD 701.00  ; ﾃﾞｰﾀ_ｼﾌﾄ
OUT TR0
AND 710.01  ; L_OV_Low_(RT1)保持
SET D10148.06
LD TR0
ANDNOT 710.01  ; L_OV_Low_(RT1)保持
RSET D10148.06
LD TR0
AND 710.02  ; L_OV_Hi_(RT1)保持
SET D10148.07
LD TR0
ANDNOT 710.02  ; L_OV_Hi_(RT1)保持
RSET D10148.07
LD TR0
AND 710.03  ; L_RV_Low_(RT1)保持
SET D10148.08
LD TR0
ANDNOT 710.03  ; L_RV_Low_(RT1)保持
RSET D10148.08
LD TR0
AND 710.04  ; L_RV_Hi_(RT1)保持
SET D10148.09
LD TR0
ANDNOT 710.04  ; L_RV_Hi_(RT1)保持
RSET D10148.09
LD TR0
AND 710.05  ; R_OV_Low_(RT1)保持
SET D10148.10
LD TR0
ANDNOT 710.05  ; R_OV_Low_(RT1)保持
RSET D10148.10

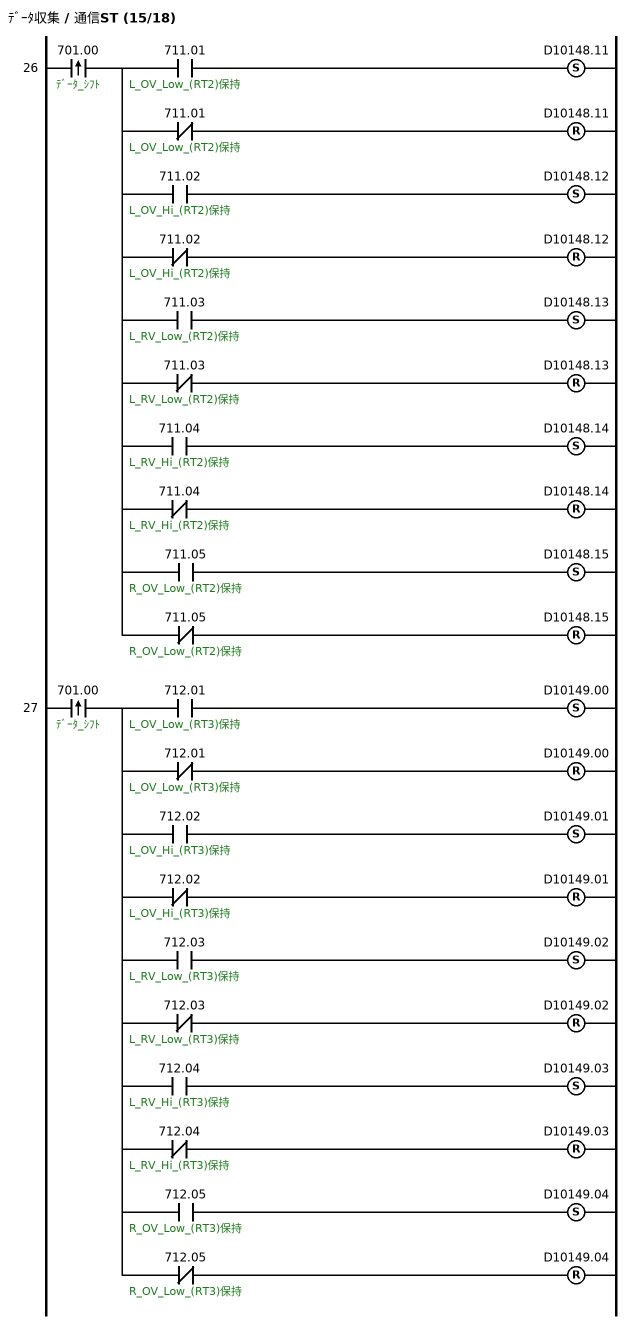
; rung 26
@LD 701.00  ; ﾃﾞｰﾀ_ｼﾌﾄ
OUT TR0
AND 711.01  ; L_OV_Low_(RT2)保持
SET D10148.11
LD TR0
ANDNOT 711.01  ; L_OV_Low_(RT2)保持
RSET D10148.11
LD TR0
AND 711.02  ; L_OV_Hi_(RT2)保持
SET D10148.12
LD TR0
ANDNOT 711.02  ; L_OV_Hi_(RT2)保持
RSET D10148.12
LD TR0
AND 711.03  ; L_RV_Low_(RT2)保持
SET D10148.13
LD TR0
ANDNOT 711.03  ; L_RV_Low_(RT2)保持
RSET D10148.13
LD TR0
AND 711.04  ; L_RV_Hi_(RT2)保持
SET D10148.14
LD TR0
ANDNOT 711.04  ; L_RV_Hi_(RT2)保持
RSET D10148.14
LD TR0
AND 711.05  ; R_OV_Low_(RT2)保持
SET D10148.15
LD TR0
ANDNOT 711.05  ; R_OV_Low_(RT2)保持
RSET D10148.15
; rung 27
@LD 701.00  ; ﾃﾞｰﾀ_ｼﾌﾄ
OUT TR0
AND 712.01  ; L_OV_Low_(RT3)保持
SET D10149.00
LD TR0
ANDNOT 712.01  ; L_OV_Low_(RT3)保持
RSET D10149.00
LD TR0
AND 712.02  ; L_OV_Hi_(RT3)保持
SET D10149.01
LD TR0
ANDNOT 712.02  ; L_OV_Hi_(RT3)保持
RSET D10149.01
LD TR0
AND 712.03  ; L_RV_Low_(RT3)保持
SET D10149.02
LD TR0
ANDNOT 712.03  ; L_RV_Low_(RT3)保持
RSET D10149.02
LD TR0
AND 712.04  ; L_RV_Hi_(RT3)保持
SET D10149.03
LD TR0
ANDNOT 712.04  ; L_RV_Hi_(RT3)保持
RSET D10149.03
LD TR0
AND 712.05  ; R_OV_Low_(RT3)保持
SET D10149.04
LD TR0
ANDNOT 712.05  ; R_OV_Low_(RT3)保持
RSET D10149.04

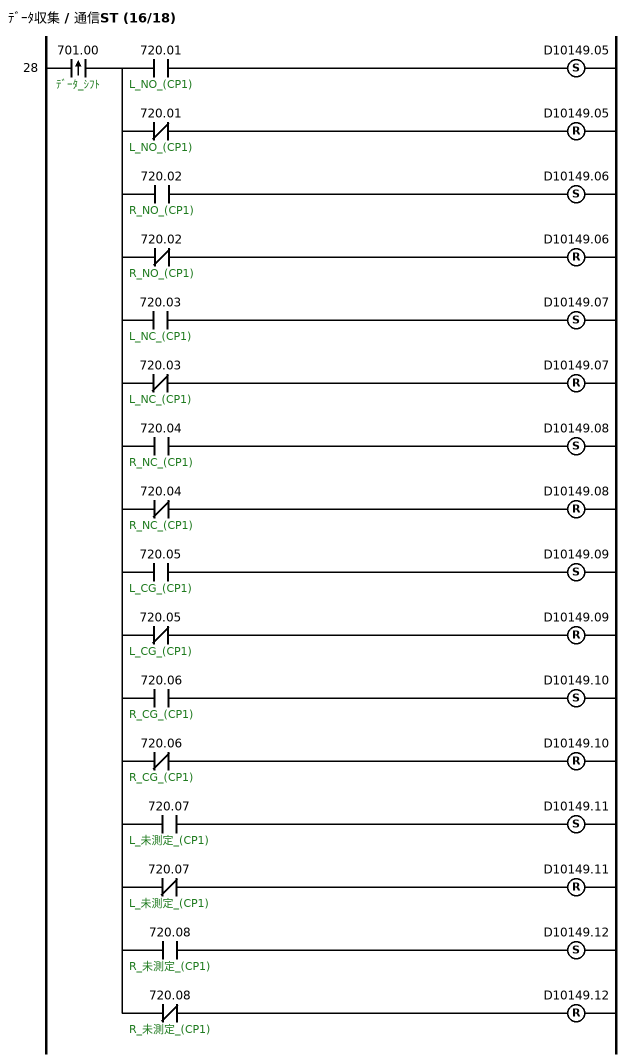
; rung 28
@LD 701.00  ; ﾃﾞｰﾀ_ｼﾌﾄ
OUT TR0
AND 720.01  ; L_NO_(CP1)
SET D10149.05
LD TR0
ANDNOT 720.01  ; L_NO_(CP1)
RSET D10149.05
LD TR0
AND 720.02  ; R_NO_(CP1)
SET D10149.06
LD TR0
ANDNOT 720.02  ; R_NO_(CP1)
RSET D10149.06
LD TR0
AND 720.03  ; L_NC_(CP1)
SET D10149.07
LD TR0
ANDNOT 720.03  ; L_NC_(CP1)
RSET D10149.07
LD TR0
AND 720.04  ; R_NC_(CP1)
SET D10149.08
LD TR0
ANDNOT 720.04  ; R_NC_(CP1)
RSET D10149.08
LD TR0
AND 720.05  ; L_CG_(CP1)
SET D10149.09
LD TR0
ANDNOT 720.05  ; L_CG_(CP1)
RSET D10149.09
LD TR0
AND 720.06  ; R_CG_(CP1)
SET D10149.10
LD TR0
ANDNOT 720.06  ; R_CG_(CP1)
RSET D10149.10
LD TR0
AND 720.07  ; L_未測定_(CP1)
SET D10149.11
LD TR0
ANDNOT 720.07  ; L_未測定_(CP1)
RSET D10149.11
LD TR0
AND 720.08  ; R_未測定_(CP1)
SET D10149.12
LD TR0
ANDNOT 720.08  ; R_未測定_(CP1)
RSET D10149.12

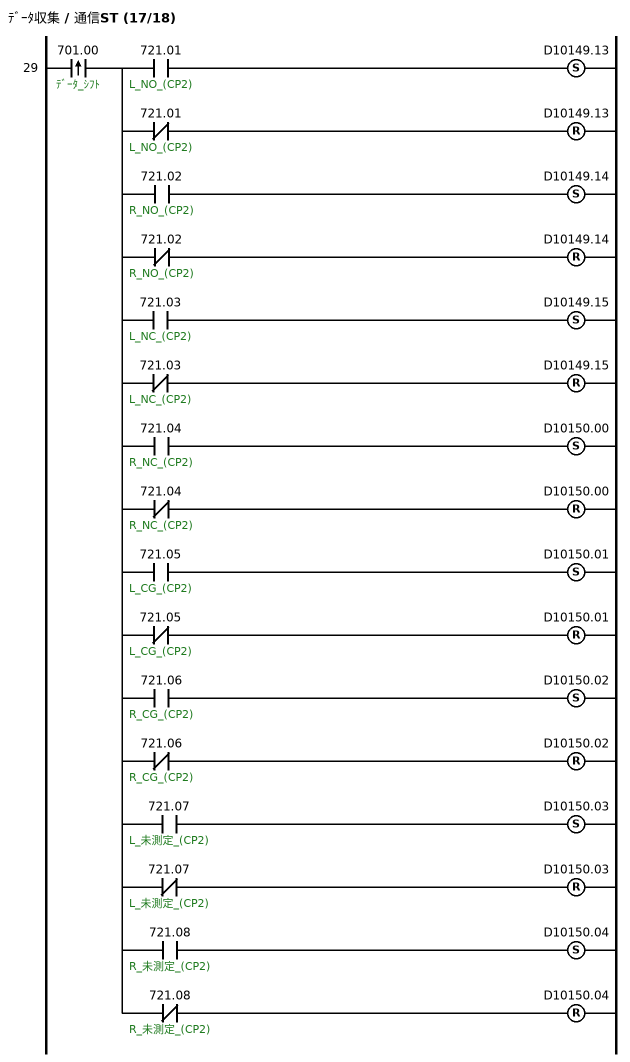
; rung 29
@LD 701.00  ; ﾃﾞｰﾀ_ｼﾌﾄ
OUT TR0
AND 721.01  ; L_NO_(CP2)
SET D10149.13
LD TR0
ANDNOT 721.01  ; L_NO_(CP2)
RSET D10149.13
LD TR0
AND 721.02  ; R_NO_(CP2)
SET D10149.14
LD TR0
ANDNOT 721.02  ; R_NO_(CP2)
RSET D10149.14
LD TR0
AND 721.03  ; L_NC_(CP2)
SET D10149.15
LD TR0
ANDNOT 721.03  ; L_NC_(CP2)
RSET D10149.15
LD TR0
AND 721.04  ; R_NC_(CP2)
SET D10150.00
LD TR0
ANDNOT 721.04  ; R_NC_(CP2)
RSET D10150.00
LD TR0
AND 721.05  ; L_CG_(CP2)
SET D10150.01
LD TR0
ANDNOT 721.05  ; L_CG_(CP2)
RSET D10150.01
LD TR0
AND 721.06  ; R_CG_(CP2)
SET D10150.02
LD TR0
ANDNOT 721.06  ; R_CG_(CP2)
RSET D10150.02
LD TR0
AND 721.07  ; L_未測定_(CP2)
SET D10150.03
LD TR0
ANDNOT 721.07  ; L_未測定_(CP2)
RSET D10150.03
LD TR0
AND 721.08  ; R_未測定_(CP2)
SET D10150.04
LD TR0
ANDNOT 721.08  ; R_未測定_(CP2)
RSET D10150.04

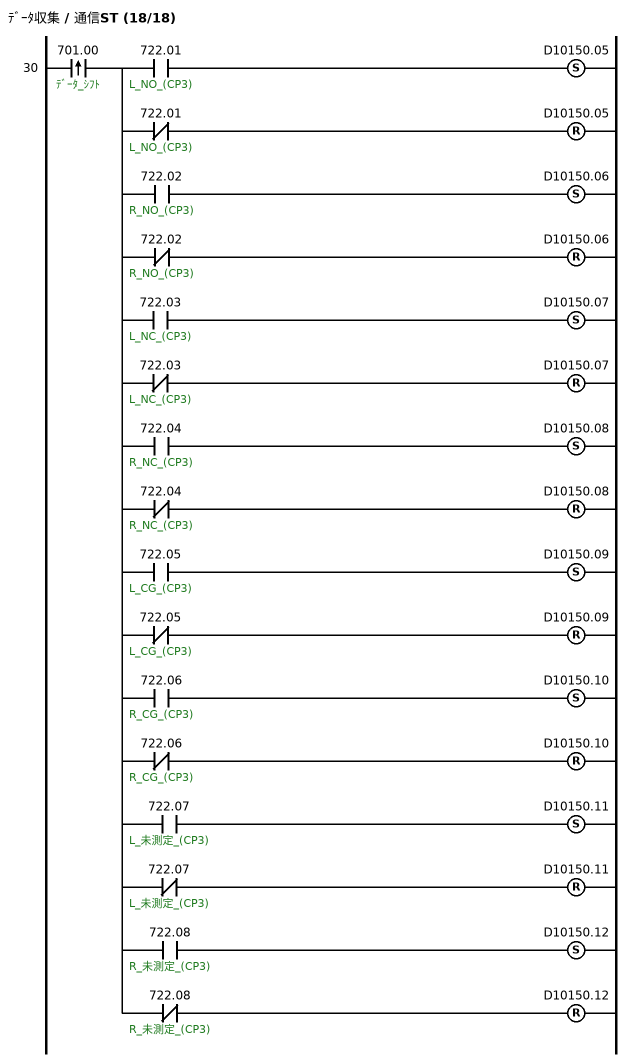
; rung 30
@LD 701.00  ; ﾃﾞｰﾀ_ｼﾌﾄ
OUT TR0
AND 722.01  ; L_NO_(CP3)
SET D10150.05
LD TR0
ANDNOT 722.01  ; L_NO_(CP3)
RSET D10150.05
LD TR0
AND 722.02  ; R_NO_(CP3)
SET D10150.06
LD TR0
ANDNOT 722.02  ; R_NO_(CP3)
RSET D10150.06
LD TR0
AND 722.03  ; L_NC_(CP3)
SET D10150.07
LD TR0
ANDNOT 722.03  ; L_NC_(CP3)
RSET D10150.07
LD TR0
AND 722.04  ; R_NC_(CP3)
SET D10150.08
LD TR0
ANDNOT 722.04  ; R_NC_(CP3)
RSET D10150.08
LD TR0
AND 722.05  ; L_CG_(CP3)
SET D10150.09
LD TR0
ANDNOT 722.05  ; L_CG_(CP3)
RSET D10150.09
LD TR0
AND 722.06  ; R_CG_(CP3)
SET D10150.10
LD TR0
ANDNOT 722.06  ; R_CG_(CP3)
RSET D10150.10
LD TR0
AND 722.07  ; L_未測定_(CP3)
SET D10150.11
LD TR0
ANDNOT 722.07  ; L_未測定_(CP3)
RSET D10150.11
LD TR0
AND 722.08  ; R_未測定_(CP3)
SET D10150.12
LD TR0
ANDNOT 722.08  ; R_未測定_(CP3)
RSET D10150.12

### Section END
; rung 0
END(001)